// TIA Portal V18 export
// export: Created 2026-06-08T17:01:58.6614111Z, ExportSetting WithDefaults, DisplayName Totally Integrated Automation Portal, DisplayVersion V18, DisplayName TIA Portal Openness, DisplayVersion V18, DisplayName TIA Portal Version Control Interface, DisplayVersion V18, DisplayName STEP 7 Professional, DisplayVersion V18, DisplayName STEP 7 Safety, DisplayVersion V18, DisplayName WinCC Professional, DisplayVersion V18
FUNCTION "DIV2_COUNTING" : Void   // FC6, LAD
{ S7_Optimized_Access := 'TRUE' }
VERSION : 0.1
// stored: AutoNumber true, IsIECCheckEnabled false, SetENOAutomatically false, UDAEnableTagReadback false
BEGIN

REGION Network 1
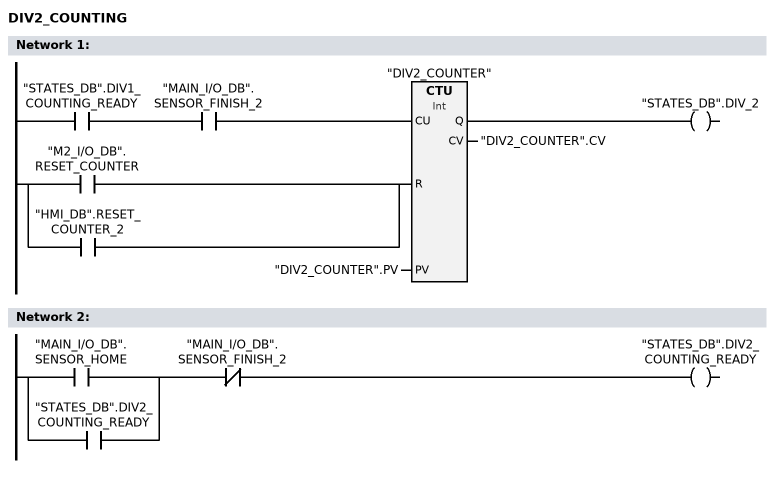
   RUNG wire#powerrail
      Contact( "STATES_DB".DIV1_COUNTING_READY )
      Contact( "MAIN_I/O_DB".SENSOR_FINISH_2 )
      { S7_Templates := "value_type := Int" } "DIV2_COUNTER".CTU(r := wire#w1, pv := "DIV2_COUNTER".PV, cv => "DIV2_COUNTER".CV)
      Coil( "STATES_DB".DIV_2 )
   END_RUNG
   RUNG wire#powerrail
      Contact( "M2_I/O_DB".RESET_COUNTER )
   END_RUNG wire#w1
   RUNG wire#powerrail
      Contact( "HMI_DB".RESET_COUNTER_2 )
   END_RUNG wire#w1
   // the same network as SCL:
   "DIV2_COUNTER".CTU(CU := "STATES_DB".DIV1_COUNTING_READY AND "MAIN_I/O_DB".SENSOR_FINISH_2,
                      R := "M2_I/O_DB".RESET_COUNTER OR "HMI_DB".RESET_COUNTER_2,
                      PV := "DIV2_COUNTER".PV,
                      CV => "DIV2_COUNTER".CV);
   "STATES_DB".DIV_2 := "DIV2_COUNTER".Q;
END_REGION

REGION Network 2
   RUNG wire#powerrail
      Contact( "MAIN_I/O_DB".SENSOR_HOME )
      wire#w1
      I_Contact( "MAIN_I/O_DB".SENSOR_FINISH_2 )
      Coil( "STATES_DB".DIV2_COUNTING_READY )
   END_RUNG
   RUNG wire#powerrail
      Contact( "STATES_DB".DIV2_COUNTING_READY )
   END_RUNG wire#w1
   // the same network as SCL:
   "STATES_DB".DIV2_COUNTING_READY := ("MAIN_I/O_DB".SENSOR_HOME OR "STATES_DB".DIV2_COUNTING_READY) AND NOT "MAIN_I/O_DB".SENSOR_FINISH_2;
END_REGION
END_FUNCTION
